Fanuc KAREL source: DOSFILE_INF.kl

PROGRAM T
%NOLOCKGROUP
VAR
 v0 : STRING[40]
 v1 : INTEGER
 v2 : STRING[40]
 v3 : INTEGER
BEGIN
 DOSFILE_INF(v0, v1, v2, v3)
END T
